TYPE ST_SixRobotActionInfo :
STRUCT
	A_Done		:BOOL;
	B_Done		:BOOL;
END_STRUCT
END_TYPE

(* stored: Version 1.1.0.1, ProductVersion 3.1.4024.13
   DUT ST_SixRobotActionInfo: Id {18396b74-e4b2-43dd-8e58-0841b29c637e} *)
